{attribute 'qualified_only'}
VAR_GLOBAL
	FQM:SensorFQM;
END_VAR

(* stored: Version 1.1.0.1, ProductVersion 3.1.4024.9
   GVL GVL: Id {adc93768-8f60-4b7a-b85c-84e47f627266} *)
